// SIMATIC S7-200 project (STEP 7-Micro/WIN), CPU 224 REL 01.11

SYMBOL_TABLE USER1
Start            I0.0
Stopp            I0.1
Xanh1            Q0.0
Vang1            Q0.1
Do1              Q0.2
Xanh2            Q0.7
Vang2            Q1.0
Do2              Q1.1
END_SYMBOL_TABLE

ORGANIZATION_BLOCK MAIN:OB1
TITLE=PROGRAM COMMENTS
BEGIN
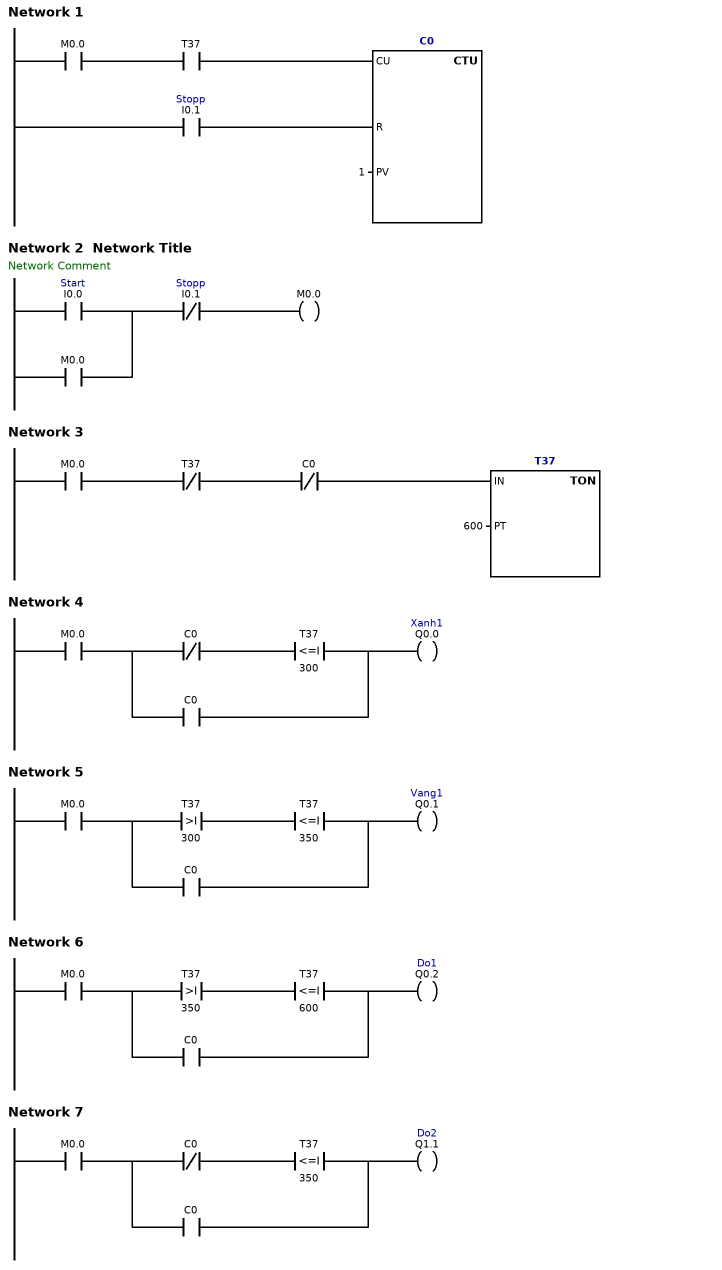
Network 1
// (network saved uncompiled; LAD cells follow)
// row 0: c0 -| |- M0.0  c1 -| |- T37  c2 --  c3 [CTU C0 CU:=power@row0, R:=power@row1, PV:=1]
// row 1: c0 --  c1 -| |- Stopp:I0.1  c2 --  c3 [box]
// row 2: c3 [box]
Network 2 // Network Title
// Network Comment
LD     Start:I0.0
O      M0.0
AN     Stopp:I0.1
=      M0.0
Network 3
LD     M0.0
AN     T37
AN     C0
TON    T37, 600
Network 4
LD     M0.0
LDN    C0
AW<=   T37, 300
O      C0
ALD
=      Xanh1:Q0.0
Network 5
LD     M0.0
LDW>   T37, 300
AW<=   T37, 350
O      C0
ALD
=      Vang1:Q0.1
Network 6
LD     M0.0
LDW>   T37, 350
AW<=   T37, 600
O      C0
ALD
=      Do1:Q0.2
Network 7
LD     M0.0
LDN    C0
AW<=   T37, 350
O      C0
ALD
=      Do2:Q1.1
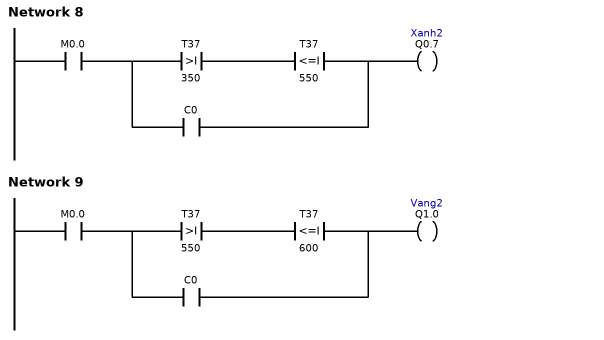
Network 8
LD     M0.0
LDW>   T37, 350
AW<=   T37, 550
O      C0
ALD
=      Xanh2:Q0.7
Network 9
LD     M0.0
LDW>   T37, 550
AW<=   T37, 600
O      C0
ALD
=      Vang2:Q1.0
END_ORGANIZATION_BLOCK
